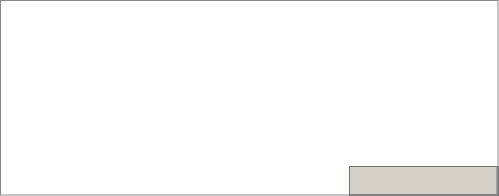
VISUALIZATION Visualization  // 499x196
    Button (349,166 150x30)
END_VISUALIZATION

(* stored: Version 1.1.0.1, ProductVersion 3.1.4024.11
   Visu Visualization: Id {32f6971d-e775-4694-a29f-4f6f97881edf} *)
